{attribute addProperty BoxType "KL2124"}
{attribute addProperty Id "Channel_1Channel_E75BD82E00Channel_2Channel_E75BD82E00Channel_3Channel_E75BD82E00Channel_4Channel_E75BD82E00"}
{attribute addProperty CRC "3323555963"}
{attribute addProperty SizeInBites "0"}
{attribute addProperty SizeInBytes "0"}
TYPE KL2124_C619707B :
STRUCT
	{attribute addProperty Name "Channel_1"}
	Channel_1 : Channel_E75BD82E;
	{attribute addProperty Name "Channel_2"}
	Channel_2 : Channel_E75BD82E;
	{attribute addProperty Name "Channel_3"}
	Channel_3 : Channel_E75BD82E;
	{attribute addProperty Name "Channel_4"}
	Channel_4 : Channel_E75BD82E;
END_STRUCT
END_TYPE

(* stored: Version 1.2.0.0, ProductVersion 3.1.4024.9
   DUT KL2124_C619707B: Id {8beddb8d-0454-418d-bc24-85534d140a7e} *)
